# EPICS StreamDevice protocol: protocols/mb2.proto
Terminator = LF;
ExtraInput = Ignore;
ReplyTimeout = 1000;

getCState {
	out "cstate";
	in "STX %d %*d %*d %(\$1)d %*d";
}
